TYPE st_IOT_params :
STRUCT
	b_controlEnable			: 	BOOL := FALSE;
	r_UpdateTimeFast		: 	REAL := 15; //seconds
	r_UpdateTimeSlow		: 	REAL := 60; //seconds
	IotCommVersion			: 	eIotCommVersion;
	DefaultLoggingBudget	:	UINT	:= 100;
END_STRUCT
END_TYPE

(* stored: Version 1.1.0.1, ProductVersion 3.1.4026.18
   DUT st_IOT_params: Id {d02d8590-bfb6-480d-8fb8-c41378cdf80b} *)
